REGION Network 3: PID-Pump_1
   #_w1 := "PID_State_Param".PID_Pump1.bModeActivate AND NOT "2_MTrig";   // rising edge
   "2_MTrig" := "PID_State_Param".PID_Pump1.bModeActivate;
   "PID_Compact_Pump-1"(Setpoint := "DB2_HMI_SET"."rSetPump-1_OUT",   // PID_Compact
                        Input := "AI_DB".PT_01.rAI_Value,
                        Reset := NOT "bStartWork_Main",
                        ModeActivate := #_w1,
                        Mode := "PID_State_Param".PID_Pump1.iModeNum,
                        Output => "Pumps".Pump_1.rAutoSpeedPump,
                        State => "PID_State_Param".PID_Pump1.iOutState,
                        Error => "PID_State_Param".PID_Pump1.bOutError,
                        ErrorBits => "PID_State_Param".PID_Pump1.iOutErrorBits);
END_REGION

REGION Network 4 (SCL): Выбор уставки для ПИД насоса - 1
   REGION Parameters PID

      // "PID_Compact_Pump-1".Config.InvertControl := TRUE;

   (* "PID_Compact_Zone1".sRet.r_Ctrl_Gain := "DB2_HMI_SET".k_PID_Zona1.Gain; // Изменение коэф. П
    "PID_Compact_Zone1".sRet.r_Ctrl_Ti  := "DB2_HMI_SET".k_PID_Zona1.I; // Изменение коэф И
    "PID_Compact_Zone1".sRet.r_Ctrl_Td  := "DB2_HMI_SET".k_PID_Zona1.D; // Изменение коэф Д
    *)
    // % Reading Tuning process
       "PID_State_Param".PID_Pump1.iProgress := "PID_Compact_Pump-1".Progress;
   END_REGION



   //Передача уставки в ПИД в зависимости от выбранного режима работы
   IF "bPosition_Diarator" THEN
       "DB2_HMI_SET"."rSetPump-1_OUT" := "DB2_HMI_SET"."rSetPump-1_Diarator";
   ELSE
       "DB2_HMI_SET"."rSetPump-1_OUT" := "DB2_HMI_SET"."rSetPump-1_CIP";
   END_IF;
END_REGION

REGION Network 5: ПИД - насос 2
   #_w1 := "PID_State_Param".PID_Pump2.bModeActivate AND NOT "3_MTrig";   // rising edge
   "3_MTrig" := "PID_State_Param".PID_Pump2.bModeActivate;
   "PID_Compact_Pump-2"(Setpoint := "DB2_HMI_SET"."rSetPump-2_OUT",   // PID_Compact
                        Input := "AI_DB".PT_03.rAI_Value,
                        Reset := NOT "bStartWork_Main",
                        ModeActivate := #_w1,
                        Mode := "PID_State_Param".PID_Pump2.iModeNum,
                        Output => "Pumps".Pump_2.rAutoSpeedPump,
                        State => "PID_State_Param".PID_Pump2.iOutState,
                        Error => "PID_State_Param".PID_Pump2.bOutError,
                        ErrorBits => "PID_State_Param".PID_Pump2.iOutErrorBits);
END_REGION

REGION Network 6 (SCL): Выбор уставки для ПИД насоса - 2
   REGION Parameters PID
       (*"
    PID_Compact_Valve_2".sPid_Cmpt.b_InvCtrl := "bTypePID_Zone1";
    "PID_Compact_Zone1".sRet.r_Ctrl_Gain := "DB2_HMI_SET".k_PID_Zona1.Gain; // Изменение коэф. П
    "PID_Compact_Zone1".sRet.r_Ctrl_Ti  := "DB2_HMI_SET".k_PID_Zona1.I; // Изменение коэф И
    "PID_Compact_Zone1".sRet.r_Ctrl_Td  := "DB2_HMI_SET".k_PID_Zona1.D; // Изменение коэф Д
    *)
    // % Reading Tuning process

   END_REGION
   "PID_State_Param".PID_Pump2.iProgress := "PID_Compact_Pump-2".Progress;
   //Передача уставки в ПИД в зависимости от выбранного режима работы
   IF "bPosition_Diarator" THEN
       "DB2_HMI_SET"."rSetPump-2_OUT" := "DB2_HMI_SET"."rSetPump-2_Diarator";
   ELSE
       "DB2_HMI_SET"."rSetPump-2_OUT" := "DB2_HMI_SET"."rSetPump-2_CIP";
   END_IF;
END_REGION
END_ORGANIZATION_BLOCK

ORGANIZATION_BLOCK "Cyclic interrupt(SCL)"   // OB32, SCL, CyclicInterrupt
{ S7_Optimized_Access := 'TRUE' }
VERSION : 0.1
   VAR_INPUT
      Initial_Call : Bool;   // Initial call of this OB
      Event_Count : Int;   // Events discarded
   END_VAR
   VAR_TEMP
      Reset : Bool;   // Сброс счетчика
   END_VAR
BEGIN
   //Условие включения накопления времени наработки установки (в свойствах ОВ - запуск каждую 1 секунду)
   //Если установка запущена и расход воды больше 1000
   //
   IF "bStartWork_Main" AND "AI_DB".FIC.rAI_Value > 500 THEN
       "diAccumTime" := "diAccumTime" + 1;     // 1 - 1 секунда, запуск ОВ жестко прописан в свойствах ОВ
   END_IF;

   //При необходимости сбросить наккопленную наработку
   //
   "R_trig_ResTimeWorkSystem"(In:="bResTimeWorkSystem",
                              Q=>#Reset);

   IF #Reset THEN
       "diAccumTime" := 0;
   END_IF;

   //Перевод накопленного времени в часы, минуты, секунды
       "iOurs_WorkSystem" := "diAccumTime" / 3600;
       "iMini_WorkSystem" := ("diAccumTime" MOD 3600) / 60;
       "iSec_WorkSystem" := "diAccumTime" MOD 60;
END_ORGANIZATION_BLOCK

ORGANIZATION_BLOCK "Исполнительные устройств"   // OB123, LAD, ProgramCycle
TITLE = Работа физических устройств
{ S7_Optimized_Access := 'TRUE' }
VERSION : 0.1
// Насосы, клапана, и т.д.
   VAR_INPUT
      Initial_Call : Bool;   // Initial call of this OB
      Remanence : Bool;   // =True, if remanent data are available
   END_VAR
BEGIN

REGION Network 1: Аналогвые датчики
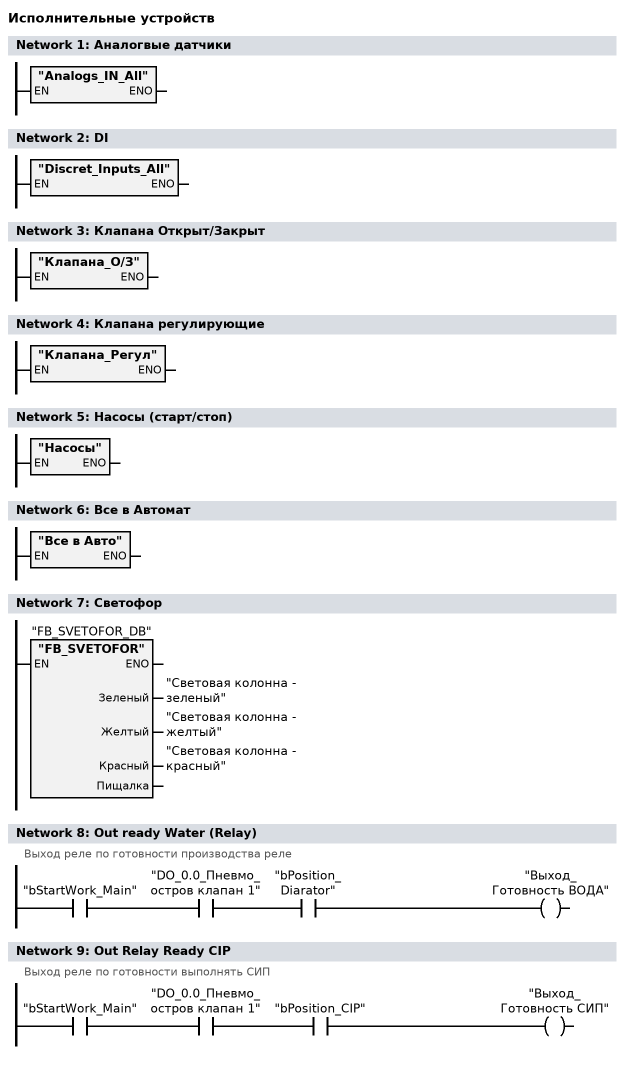
   RUNG wire#powerrail
      "Analogs_IN_All"()
   END_RUNG
   // the same network as SCL:
   "Analogs_IN_All"();
END_REGION

REGION Network 2: DI
   RUNG wire#powerrail
      "Discret_Inputs_All"()
   END_RUNG
   // the same network as SCL:
   "Discret_Inputs_All"();
END_REGION

REGION Network 3: Клапана Открыт/Закрыт
   RUNG wire#powerrail
      "Клапана_О/З"()
   END_RUNG
   // the same network as SCL:
   "Клапана_О/З"();
END_REGION

REGION Network 4: Клапана регулирующие
   RUNG wire#powerrail
      "Клапана_Регул"()
   END_RUNG
   // the same network as SCL:
   "Клапана_Регул"();
END_REGION

REGION Network 5: Насосы (старт/стоп)
   RUNG wire#powerrail
      "Насосы"()
   END_RUNG
   // the same network as SCL:
   "Насосы"();
END_REGION

REGION Network 6: Все в Автомат
   RUNG wire#powerrail
      "Все в Авто"()
   END_RUNG
   // the same network as SCL:
   "Все в Авто"();
END_REGION

REGION Network 7: Светофор
   RUNG wire#powerrail
      "FB_SVETOFOR_DB"(Зеленый => "Световая колонна - зеленый", Желтый => "Световая колонна - желтый", Красный => "Световая колонна - красный", Пищалка =>)
   END_RUNG
   // the same network as SCL:
   "FB_SVETOFOR_DB"(Зеленый => "Световая колонна - зеленый",   // "FB_SVETOFOR"
                    Желтый => "Световая колонна - желтый",
                    Красный => "Световая колонна - красный");
END_REGION

REGION Network 8: Out ready Water (Relay)
   // Выход реле по готовности производства реле
   RUNG wire#powerrail
      Contact( "bStartWork_Main" )
      Contact( "DO_0.0_Пневмо_остров клапан 1" )
      Contact( "bPosition_Diarator" )
      Coil( "Выход_Готовность ВОДА" )
   END_RUNG
   // the same network as SCL:
   "Выход_Готовность ВОДА" := "bStartWork_Main" AND "DO_0.0_Пневмо_остров клапан 1" AND "bPosition_Diarator";
END_REGION

REGION Network 9: Out Relay Ready CIP
   // Выход реле по готовности выполнять СИП
   RUNG wire#powerrail
      Contact( "bStartWork_Main" )
      Contact( "DO_0.0_Пневмо_остров клапан 1" )
      Contact( "bPosition_CIP" )
      Coil( "Выход_Готовность СИП" )
   END_RUNG
   // the same network as SCL:
   "Выход_Готовность СИП" := "bStartWork_Main" AND "DO_0.0_Пневмо_остров клапан 1" AND "bPosition_CIP";
END_REGION
END_ORGANIZATION_BLOCK

ORGANIZATION_BLOCK "Counters"   // OB125, LAD, ProgramCycle
TITLE = "Main Program Sweep (Cycle)"
{ S7_Optimized_Access := 'TRUE' }
VERSION : 0.1
// Различные счетчики
   VAR_INPUT
      Initial_Call : Bool;   // Initial call of this OB
      Remanence : Bool;   // =True, if remanent data are available
   END_VAR
   VAR_TEMP   // added for the SCL form of the ladder/FBD networks
      _w1 : Bool;
      _w2 : Bool;
   END_VAR
BEGIN

REGION Network 1: Counter Water to Sewerage
   // Счетчик сброшенной воды в канализацию
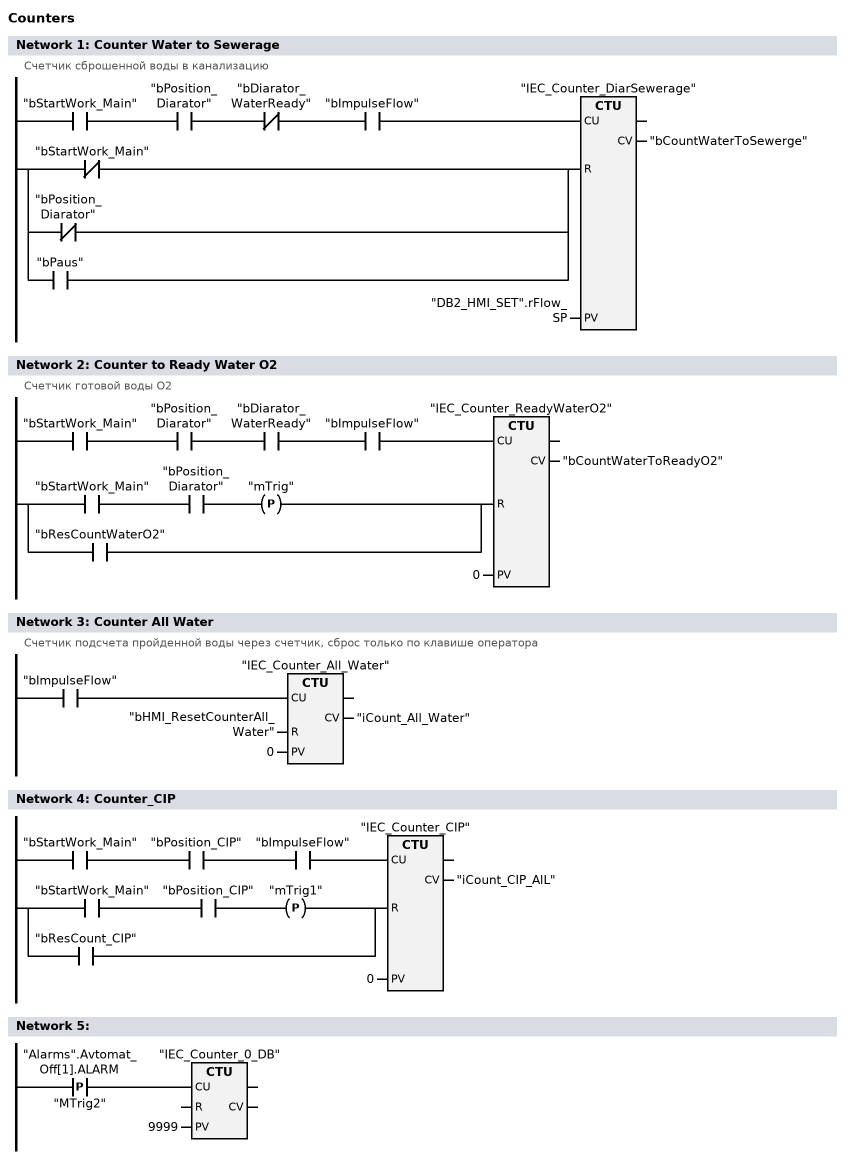
   "IEC_Counter_DiarSewerage".CTU(CU := "bStartWork_Main" AND "bPosition_Diarator" AND NOT "bDiarator_WaterReady" AND "bImpulseFlow",
                           R := NOT "bStartWork_Main" OR NOT "bPosition_Diarator" OR "bPaus",
                           PV := "DB2_HMI_SET".rFlow_SP,
                           CV => "bCountWaterToSewerge");
END_REGION

REGION Network 2: Counter to Ready Water O2
   // Счетчик готовой воды О2
   #_w1 := "bStartWork_Main" AND "bPosition_Diarator";
   #_w2 := #_w1 AND NOT "mTrig";   // rising edge
   "mTrig" := #_w1;
   "IEC_Counter_ReadyWaterO2".CTU(CU := "bStartWork_Main" AND "bPosition_Diarator" AND "bDiarator_WaterReady" AND "bImpulseFlow",
                           R := #_w2 OR "bResCountWaterO2",
                           PV := 0,
                           CV => "bCountWaterToReadyO2");
END_REGION

REGION Network 3: Counter All Water
   // Счетчик подсчета пройденной воды через счетчик, сброс только по клавише оператора
   "IEC_Counter_All_Water".CTU(CU := "bImpulseFlow",
                           R := "bHMI_ResetCounterAll_Water",
                           PV := 0,
                           CV => "iCount_All_Water");
END_REGION

REGION Network 4: Counter_CIP
   #_w1 := "bStartWork_Main" AND "bPosition_CIP";
   #_w2 := #_w1 AND NOT "mTrig1";   // rising edge
   "mTrig1" := #_w1;
   "IEC_Counter_CIP".CTU(CU := "bStartWork_Main" AND "bPosition_CIP" AND "bImpulseFlow",
                         R := #_w2 OR "bResCount_CIP",
                         PV := 0,
                         CV => "iCount_CIP_AlL");
END_REGION

REGION Network 5
   #_w1 := "Alarms".Avtomat_Off[1].ALARM AND NOT "MTrig2";   // rising edge of "Alarms".Avtomat_Off[1].ALARM
   "MTrig2" := "Alarms".Avtomat_Off[1].ALARM;
   "IEC_Counter_0_DB".CTU(CU := #_w1, PV := 9999);
END_REGION
END_ORGANIZATION_BLOCK

// folder: AI_Signal

FUNCTION_BLOCK "AI_(4-20)_1"   // FB13, LAD
{ S7_Optimized_Access := 'FALSE' }
VERSION : 0.1
   VAR_INPUT
      Input_PLC : Int;   // Вход_Значение на ПЛК
      "HMI_Simulate_on/off" : Bool;   // 0 - выкл, 1 - вкл
      HMI_rSimulate_value : Real;   // значение
      HMI_rParam_Sensor_HL : Real := 16.0;   // Параметры датчика по паспорту (макс значение)bar, C, итд
      HMI_rParam_Sensor_LL : Real;   // Параметры датчика по паспорту (мин значение)bar, C, итд
      "HMI_Filtr_On/off" : Bool;   // Фильтрация, true - вкл
   END_VAR
   VAR_OUTPUT
      HMI_Value_OUT : Real;   // Значение в ед. измерения
      Error_out : Bool;   // Ошибка датчика
   END_VAR
   VAR
      OUT_Scale : Real;   // Выход скалированного значения
      OUT_Normal_Ed : Real;   // Выход нормализованной единицы от 0 др 1
      AI_filtr : "AI_Filtr";
      HMI_Range : Int := 10;   // Кол-во данных для фильтрации
      HMI_iSet_Tik : Int := 2;   // Скорость набора данных для фильтрации
   END_VAR
   VAR_TEMP
      Input_PLC_to_dint : DInt;   // Конвертация из инт в реал
      Error : Word;   // Ошибка в скалировании
      "PLC to_real" : Real;
      value_scale : Real;
      Input_PLC_temp : Int;
      OFF_Param : Bool;
   END_VAR
BEGIN

REGION Network 1
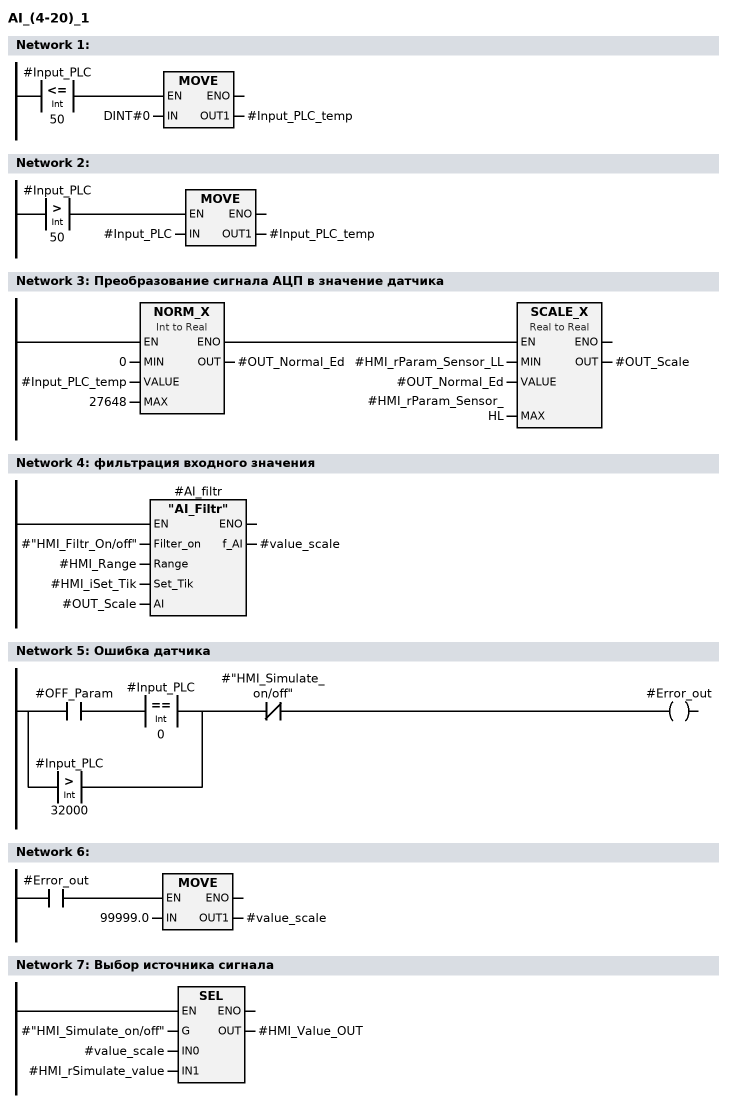
   RUNG wire#powerrail
      { S7_Templates := "SrcType := Int" } LE_Contact(in1 := #Input_PLC, in2 := 50)
      { S7_GenerateENO := "TRUE" } Move(in := DINT#0, out1 => #Input_PLC_temp)
   END_RUNG
   // the same network as SCL:
   IF #Input_PLC <= 50 THEN #Input_PLC_temp := DINT#0; END_IF;
END_REGION

REGION Network 2
   RUNG wire#powerrail
      { S7_Templates := "SrcType := Int" } GT_Contact(in1 := #Input_PLC, in2 := 50)
      { S7_GenerateENO := "TRUE" } Move(in := #Input_PLC, out1 => #Input_PLC_temp)
   END_RUNG
   // the same network as SCL:
   IF #Input_PLC > 50 THEN #Input_PLC_temp := #Input_PLC; END_IF;
END_REGION

REGION Network 3: Преобразование сигнала АЦП в значение датчика
   RUNG wire#powerrail
      { S7_Templates := "[SrcType := Int, DestType := Real]" } Normalize(min := 0, value := #Input_PLC_temp, max := 27648, out => #OUT_Normal_Ed)
      { S7_Templates := "[SrcType := Real, DestType := Real]" } Scale(min := #HMI_rParam_Sensor_LL, value := #OUT_Normal_Ed, max := #HMI_rParam_Sensor_HL, out => #OUT_Scale)
   END_RUNG
   // the same network as SCL:
   #OUT_Normal_Ed := NORM_X(MIN := 0, VALUE := #Input_PLC_temp, MAX := 27648);
   #OUT_Scale := SCALE_X(MIN := #HMI_rParam_Sensor_LL, VALUE := #OUT_Normal_Ed, MAX := #HMI_rParam_Sensor_HL);
END_REGION

REGION Network 4: фильтрация входного значения
   RUNG wire#powerrail
      #AI_filtr(Filter_on := #"HMI_Filtr_On/off", Range := #HMI_Range, Set_Tik := #HMI_iSet_Tik, AI := #OUT_Scale, f_AI => #value_scale)
   END_RUNG
   // the same network as SCL:
   #AI_filtr(Filter_on := #"HMI_Filtr_On/off",   // "AI_Filtr"
             Range := #HMI_Range,
             Set_Tik := #HMI_iSet_Tik,
             AI := #OUT_Scale,
             f_AI => #value_scale);
END_REGION

REGION Network 5: Ошибка датчика
   RUNG wire#powerrail
      Contact( #OFF_Param )
      { S7_Templates := "SrcType := Int" } EQ_Contact(in1 := #Input_PLC, in2 := 0)
      wire#w1
      I_Contact( #"HMI_Simulate_on/off" )
      Coil( #Error_out )
   END_RUNG
   RUNG wire#powerrail
      { S7_Templates := "SrcType := Int" } GT_Contact(in1 := #Input_PLC, in2 := 32000)
   END_RUNG wire#w1
   // the same network as SCL:
   #Error_out := ((#OFF_Param AND (#Input_PLC = 0)) OR (#Input_PLC > 32000)) AND NOT #"HMI_Simulate_on/off";
END_REGION

REGION Network 6
   RUNG wire#powerrail
      Contact( #Error_out )
      Move(in := 99999.0, out1 => #value_scale)
   END_RUNG
   // the same network as SCL:
   IF #Error_out THEN #value_scale := 99999.0; END_IF;
END_REGION

REGION Network 7: Выбор источника сигнала
   #HMI_Value_OUT := SEL(G := #"HMI_Simulate_on/off", IN0 := #value_scale, IN1 := #HMI_rSimulate_value);
END_REGION
END_FUNCTION_BLOCK

FUNCTION_BLOCK "AI_(PT100)"   // FB21, LAD
{ S7_Optimized_Access := 'FALSE' }
VERSION : 0.1
   VAR_INPUT
      Input_PLC : Int;   // Вход_Значение на ПЛК
      "Simulate_on/off" : Bool;   // 0 - выкл, 1 - вкл
      Simulate_value : Real;   // значение
      Param_Sensor_HL : Real := 16.0;   // Параметры датчика по паспорту (макс значение)bar, C, итд
      Param_Sensor_LL : Real;   // Параметры датчика по паспорту (мин значение)bar, C, итд
      "Filtr_On/off" : Bool;   // Фильтрация, true - вкл
   END_VAR
   VAR_OUTPUT
      Value_OUT : Real;   // Значение в ед. измерения
      Error_out : Bool;   // Ошибка датчика
   END_VAR
   VAR
      bipolar : Bool;
      OUT_Scale : Real;   // Выход скалированного значения
      AI_filtr : "AI_Filtr";
      Range : Int := 10;   // Кол-во данных для фильтрации
   END_VAR
   VAR_TEMP
      Input_PLC_to_dint : DInt;   // Конвертация из инт в реал
      Error : Word;   // Ошибка в скалировании
      "PLC to_real" : Real;
      value_scale : Real;
      Input_PLC_temp : Int;
      Input_PLC_to_real : Real;
   END_VAR
BEGIN

REGION Network 1
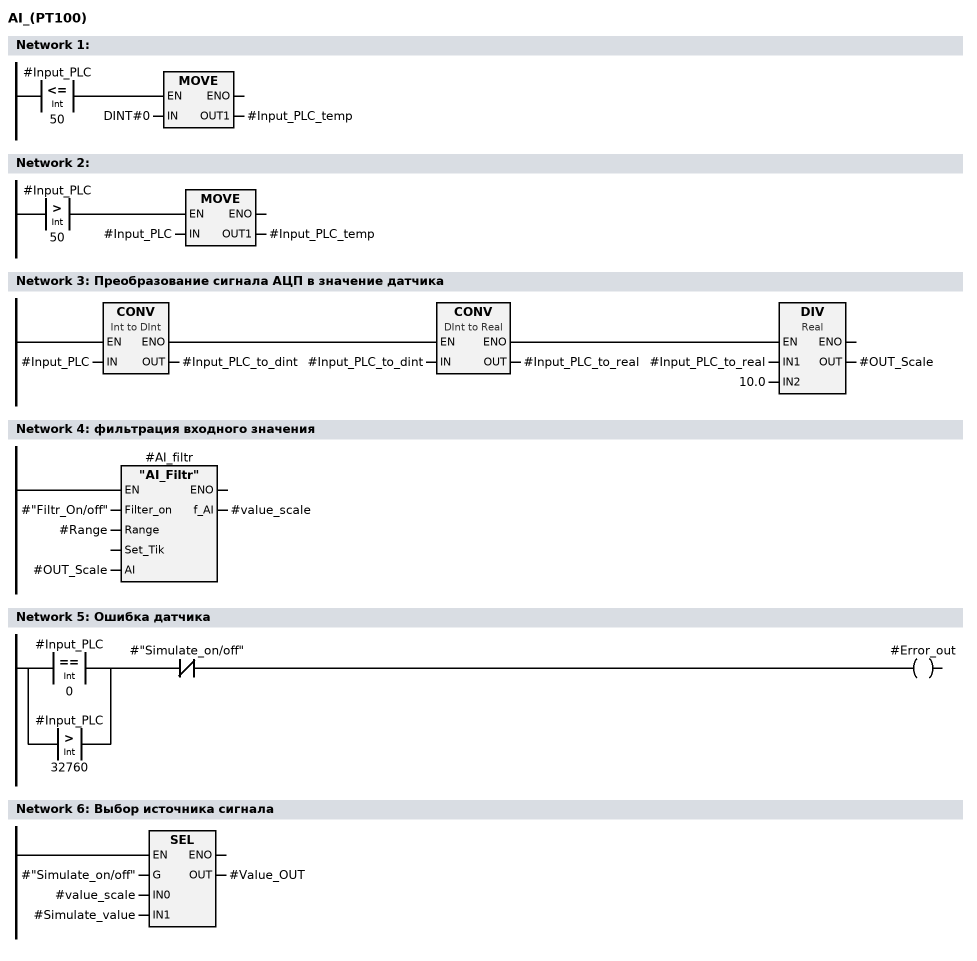
   RUNG wire#powerrail
      { S7_Templates := "SrcType := Int" } LE_Contact(in1 := #Input_PLC, in2 := 50)
      { S7_GenerateENO := "TRUE" } Move(in := DINT#0, out1 => #Input_PLC_temp)
   END_RUNG
   // the same network as SCL:
   IF #Input_PLC <= 50 THEN #Input_PLC_temp := DINT#0; END_IF;
END_REGION

REGION Network 2
   RUNG wire#powerrail
      { S7_Templates := "SrcType := Int" } GT_Contact(in1 := #Input_PLC, in2 := 50)
      { S7_GenerateENO := "TRUE" } Move(in := #Input_PLC, out1 => #Input_PLC_temp)
   END_RUNG
   // the same network as SCL:
   IF #Input_PLC > 50 THEN #Input_PLC_temp := #Input_PLC; END_IF;
END_REGION

REGION Network 3: Преобразование сигнала АЦП в значение датчика
   RUNG wire#powerrail
      { S7_Templates := "[SrcType := Int, DestType := DInt]"; S7_GenerateENO := "TRUE" } Convert(in := #Input_PLC, out => #Input_PLC_to_dint)
      { S7_Templates := "[SrcType := DInt, DestType := Real]"; S7_GenerateENO := "TRUE" } Convert(in := #Input_PLC_to_dint, out => #Input_PLC_to_real)
      { S7_Templates := "SrcType := Real"; S7_GenerateENO := "TRUE" } Div(in1 := #Input_PLC_to_real, in2 := 10.0, out => #OUT_Scale)
   END_RUNG
   // the same network as SCL:
   // ENO of a box is taken as its EN; it also drops when the box reports an error
   #Input_PLC_to_dint := INT_TO_DINT(#Input_PLC);
   #Input_PLC_to_real := DINT_TO_REAL(#Input_PLC_to_dint);
   #OUT_Scale := #Input_PLC_to_real / 10.0;
END_REGION

REGION Network 4: фильтрация входного значения
   RUNG wire#powerrail
      #AI_filtr(Filter_on := #"Filtr_On/off", Range := #Range, Set_Tik :=, AI := #OUT_Scale, f_AI => #value_scale)
   END_RUNG
   // the same network as SCL:
   #AI_filtr(Filter_on := #"Filtr_On/off", Range := #Range, AI := #OUT_Scale, f_AI => #value_scale);   // "AI_Filtr"
END_REGION

REGION Network 5: Ошибка датчика
   RUNG wire#powerrail
      { S7_Templates := "SrcType := Int" } EQ_Contact(in1 := #Input_PLC, in2 := 0)
      wire#w1
      I_Contact( #"Simulate_on/off" )
      Coil( #Error_out )
   END_RUNG
   RUNG wire#powerrail
      { S7_Templates := "SrcType := Int" } GT_Contact(in1 := #Input_PLC, in2 := 32760)
   END_RUNG wire#w1
   // the same network as SCL:
   #Error_out := ((#Input_PLC = 0) OR (#Input_PLC > 32760)) AND NOT #"Simulate_on/off";
END_REGION

REGION Network 6: Выбор источника сигнала
   #Value_OUT := SEL(G := #"Simulate_on/off", IN0 := #value_scale, IN1 := #Simulate_value);
END_REGION
END_FUNCTION_BLOCK

// folder: AI_Signal/Funktion

FUNCTION_BLOCK "AI_Filtr"   // FB14, SCL
{ S7_Optimized_Access := 'FALSE' }
VERSION : 0.1
   VAR_INPUT
      Filter_on : Bool;   // Вкл фильтрации
      Range : Int := 10;   // Кол-во входных значений для вычисления среднего
      Set_Tik : Int := 6;   // Задача периода фильтрации от 1(мин) до 8
      AI : Real;   // Вход значения датчика
   END_VAR
   VAR_OUTPUT
      f_AI : Real;   // выход значения с фильтром или без
   END_VAR
   VAR
      CTU : CTU_INT;   // счетчик для подсчета кол-во вх значений
      Tik : Bool;   // Время фильтрации
      ai_array : Array[0..#Max_Array] of Real;   // Массив значений датчика
      i : Int;   // для цикла ФОР
      sum_AI : Real;   // Суммирование значений с входа датчика
      Avarage_AI : Real;   // Среднее значение датчика
      fRS_set : Bool;   // Для RS тригера
      fRS_res : Bool;   // Для RS тригера
      fRS_out : Bool;   // Для RS тригера
      FullFiltr : Bool;   // Ожидание наполнения значений для вычисления средней
      Res_count : Bool;   // сброс счетчика
   END_VAR
   VAR CONSTANT
      Max_Array : Int := 30;   // Размер массива
   END_VAR
BEGIN

   CASE #Set_Tik OF                   
       1:  
           #Tik := "Time_0.1s";
       2:  
           #Tik := "Time_0.2s";
       3:
           #Tik := "Time_0.4s";
       4:
           #Tik := "Time_0.5s";
       5:
           #Tik := "Time_0.8s";
       6:
           #Tik := "Time_1s";
       7:
           #Tik := "Time_1.6s";
       8:
           #Tik := "Time_2s";
       0:
           #Tik := "Time_0.1s";

       ELSE  
           #Set_Tik := 8;
   END_CASE;  // Выбор периода фильтрации входного сигнала
   REGION RS триггер
       IF #fRS_set THEN
           #fRS_out := true;
       ELSIF #fRS_res AND NOT #fRS_set THEN
           #fRS_out := false;
       END_IF;
   END_REGION

   REGION Подсчет среднего значения входа
       // Statement section REGION
           #CTU(CU := #Tik,
                PV := #Range,
                R := #Res_count,
                Q => #Res_count);                                      // Счетчик для набора значений с входа
           #ai_array[#CTU.CV] := #AI;                                  // Запись значений с входа в массив

           IF #Res_count THEN                                              // СБРОС как счетчик переполниться Для корректной работы счетчика
               #i := 0;
               #sum_AI := 0;
           END_IF;

           IF #Range <> #i THEN                                    // выход из цикла FOR при суммировании всех значений, почему то сам не прекращел подсчет при окончании цикла все время суммировался 
               FOR #i := 0 TO (#Range - 1) DO
                   #sum_AI := #ai_array[#i] + #sum_AI;             // суммирование значений
               END_FOR;
           END_IF;

       #Avarage_AI := #sum_AI / #Range;                             // Вычисление среднего значения
       #fRS_res := NOT #Filter_on;

   END_REGION

   REGION Выбор выхода прямое или фильтрованное значение
       IF #Filter_on THEN                                          //Включение выключение фильтрации
           #fRS_set := #CTU.QD;                                    //При включении фильтра ждем наполнения значениями с входа, пока ждем - отправляем на выход прямое значение входа, далее фильтруем
            #FullFiltr := #fRS_out;

          IF #FullFiltr THEN                                       //Когда фильтр наполнился - вывыодим среднее значение входа
               #f_AI := #Avarage_AI;                              // ЗАпись значения на выход AI
          ELSE
               #f_AI := #AI;                                     // Прямой вывод значения, пока значения не наполнились данными
          END_IF;
       ELSE
           #f_AI := #AI;                                        // Если фильтр выключен, на выход прямое значение с входа
       END_IF; 

   END_REGION
END_FUNCTION_BLOCK

FUNCTION "Calculate_AI" : Void   // FC7, SCL
{ S7_Optimized_Access := 'FALSE' }
VERSION : 0.1
   VAR_INPUT
      IN_sensors : Int;
      Current_max : Real;
      Current_min : Real;
      Code_HL : Real;
      Code_LL : Real;
      Param_Sensor_HL : Real;   // Параметры датчика по паспорту (макс значение)bar, C, итд
      Param_Sensor_LL : Real;   // Параметры датчика по паспорту (мин значение)bar, C, итд
   END_VAR
   VAR_OUTPUT
      signal_Electric : Real;   // выход в электрических ед измерения
      Value_Sensor : Real;   // выход реального значения датчика в ед измерения
   END_VAR
   VAR_TEMP
      sensor_to_real : Real;   // Для конвертации INT to Real
      result_to_out_signal : Real;   // Для вычитания реального значения показания датчика
   END_VAR
BEGIN
       //Convert int to real
   #sensor_to_real := INT_TO_REAL(#IN_sensors);

       // Расчет значения АЦП контроллера в значение эл. ед измерения (I, U) в зависимости от значений на входе
   #signal_Electric := ((#sensor_to_real - #Code_LL) * (#Current_max - #Current_min) / (#Code_HL - #Code_LL))+ #Current_min;
   #result_to_out_signal := #signal_Electric;

   // Расчет значения в реальных единицах измерения датчика (bar, C,) в зависимости от введеных параметров датчика Param_Sensor min/max
   #Value_Sensor := (#result_to_out_signal - #Current_min) * (#Param_Sensor_HL - #Param_Sensor_LL) / (#Current_max - #Current_min) + #Param_Sensor_LL;
END_FUNCTION

// folder: DI_signal

FUNCTION_BLOCK "FB_DI"   // FB15, LAD
TITLE = Блок обработки дискретных входов
{ S7_Optimized_Access := 'FALSE' }
VERSION : 0.1
   VAR_INPUT
      input_value : Bool;   // Входной тэг контроллера
      "On/Off_Filters_DI" : Bool;   // Вкл/выкл фильтрацию входа
      Set_Time_Dely : Time;   // Уставка времени фильтрации
      Simulate : Bool;   // Симуляция входа (Вкл/Выкл)
      Simulate_Value : Bool;   // Значение симуляции
   END_VAR
   VAR_OUTPUT
      Value : Bool;   // Обработанный сигнал
   END_VAR
   VAR
      Time_Delay : Time;   // Время фильтрации для таймера
      Time_On : TON_TIME;   // Фильтр на Вкл
      Time_Off : TON_TIME;   // Фильтр на Выкл
      Nul_Time : Time := T#1MS;   // Откл фильтрации (0)
   END_VAR
BEGIN

REGION Network 1: Включение фильтрации
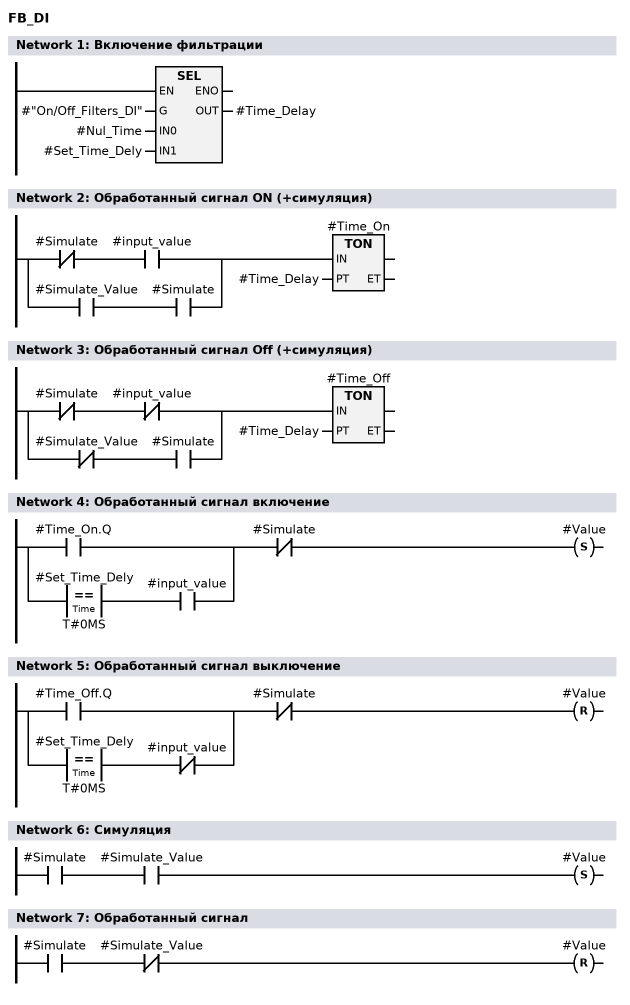
   #Time_Delay := SEL(G := #"On/Off_Filters_DI", IN0 := #Nul_Time, IN1 := #Set_Time_Dely);
END_REGION

REGION Network 2: Обработанный сигнал ON (+симуляция)
   #Time_On(IN := (NOT #Simulate AND #input_value) OR (#Simulate_Value AND #Simulate), PT := #Time_Delay);   // TON
END_REGION

REGION Network 3: Обработанный сигнал Off (+симуляция)
   #Time_Off(IN := (NOT #Simulate AND NOT #input_value) OR (NOT #Simulate_Value AND #Simulate),   // TON
             PT := #Time_Delay);
END_REGION

REGION Network 4: Обработанный сигнал включение
   RUNG wire#powerrail
      Contact( #Time_On.Q )
      wire#w1
      I_Contact( #Simulate )
      S_Coil( #Value )
   END_RUNG
   RUNG wire#powerrail
      { S7_Templates := "SrcType := Time" } EQ_Contact(in1 := #Set_Time_Dely, in2 := T#0MS)
      Contact( #input_value )
   END_RUNG wire#w1
   // the same network as SCL:
   IF (#Time_On.Q OR ((#Set_Time_Dely = T#0MS) AND #input_value)) AND NOT #Simulate THEN
       #Value := TRUE;
   END_IF;
END_REGION

REGION Network 5: Обработанный сигнал выключение
   RUNG wire#powerrail
      Contact( #Time_Off.Q )
      wire#w1
      I_Contact( #Simulate )
      R_Coil( #Value )
   END_RUNG
   RUNG wire#powerrail
      { S7_Templates := "SrcType := Time" } EQ_Contact(in1 := #Set_Time_Dely, in2 := T#0MS)
      I_Contact( #input_value )
   END_RUNG wire#w1
   // the same network as SCL:
   IF (#Time_Off.Q OR ((#Set_Time_Dely = T#0MS) AND NOT #input_value)) AND NOT #Simulate THEN
       #Value := FALSE;
   END_IF;
END_REGION

REGION Network 6: Симуляция
   RUNG wire#powerrail
      Contact( #Simulate )
      Contact( #Simulate_Value )
      S_Coil( #Value )
   END_RUNG
   // the same network as SCL:
   IF #Simulate AND #Simulate_Value THEN #Value := TRUE; END_IF;
END_REGION

REGION Network 7: Обработанный сигнал
   RUNG wire#powerrail
      Contact( #Simulate )
      I_Contact( #Simulate_Value )
      R_Coil( #Value )
   END_RUNG
   // the same network as SCL:
   IF #Simulate AND NOT #Simulate_Value THEN #Value := FALSE; END_IF;
END_REGION
END_FUNCTION_BLOCK

FUNCTION_BLOCK "FB_DI_Pointer"   // FB17, LAD
TITLE = Блок обработки дискретных входов
{ S7_Optimized_Access := 'FALSE' }
VERSION : 0.1
   VAR_INPUT
      input_value : Bool;   // Входной тэг контроллера
   END_VAR
   VAR_OUTPUT
      Value : Bool;   // Обработанный сигнал
   END_VAR
   VAR_IN_OUT
      Di_Struct : "Tipe_DI";
   END_VAR
   VAR
      Time_Delay : Time;   // Время фильтрации для таймера
      Time_On : TON_TIME;   // Фильтр на Вкл
      Time_Off : TON_TIME;   // Фильтр на Выкл
      Nul_Time : Time := T#1MS;   // Откл фильтрации (0)
      testdel : Bool;
      On_del : Bool;
   END_VAR
BEGIN

REGION Network 1: Включение фильтрации
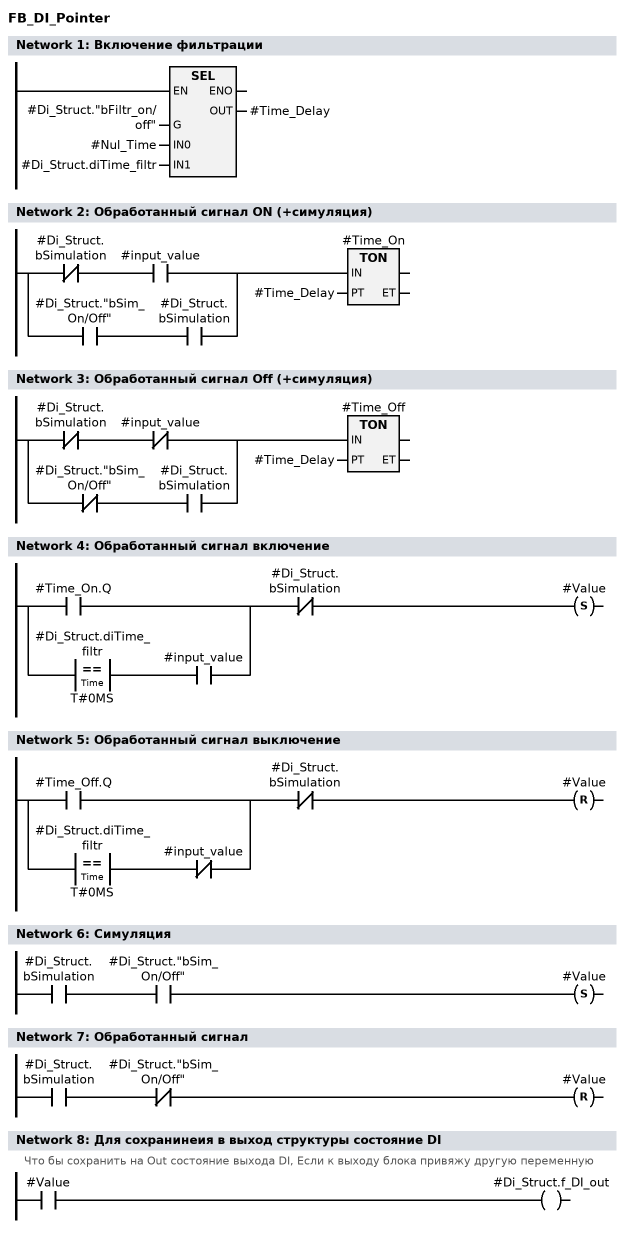
   #Time_Delay := SEL(G := #Di_Struct."bFiltr_on/off", IN0 := #Nul_Time, IN1 := #Di_Struct.diTime_filtr);
END_REGION

REGION Network 2: Обработанный сигнал ON (+симуляция)
   #Time_On(IN := (NOT #Di_Struct.bSimulation AND #input_value) OR (#Di_Struct."bSim_On/Off" AND #Di_Struct.bSimulation),   // TON
            PT := #Time_Delay);
END_REGION

REGION Network 3: Обработанный сигнал Off (+симуляция)
   #Time_Off(IN := (NOT #Di_Struct.bSimulation AND NOT #input_value) OR (NOT #Di_Struct."bSim_On/Off" AND #Di_Struct.bSimulation),   // TON
             PT := #Time_Delay);
END_REGION

REGION Network 4: Обработанный сигнал включение
   RUNG wire#powerrail
      Contact( #Time_On.Q )
      wire#w1
      I_Contact( #Di_Struct.bSimulation )
      S_Coil( #Value )
   END_RUNG
   RUNG wire#powerrail
      { S7_Templates := "SrcType := Time" } EQ_Contact(in1 := #Di_Struct.diTime_filtr, in2 := T#0MS)
      Contact( #input_value )
   END_RUNG wire#w1
   // the same network as SCL:
   IF (#Time_On.Q OR ((#Di_Struct.diTime_filtr = T#0MS) AND #input_value)) AND NOT #Di_Struct.bSimulation THEN
       #Value := TRUE;
   END_IF;
END_REGION

REGION Network 5: Обработанный сигнал выключение
   RUNG wire#powerrail
      Contact( #Time_Off.Q )
      wire#w1
      I_Contact( #Di_Struct.bSimulation )
      R_Coil( #Value )
   END_RUNG
   RUNG wire#powerrail
      { S7_Templates := "SrcType := Time" } EQ_Contact(in1 := #Di_Struct.diTime_filtr, in2 := T#0MS)
      I_Contact( #input_value )
   END_RUNG wire#w1
   // the same network as SCL:
   IF (#Time_Off.Q OR ((#Di_Struct.diTime_filtr = T#0MS) AND NOT #input_value)) AND NOT #Di_Struct.bSimulation THEN
       #Value := FALSE;
   END_IF;
END_REGION

REGION Network 6: Симуляция
   RUNG wire#powerrail
      Contact( #Di_Struct.bSimulation )
      Contact( #Di_Struct."bSim_On/Off" )
      S_Coil( #Value )
   END_RUNG
   // the same network as SCL:
   IF #Di_Struct.bSimulation AND #Di_Struct."bSim_On/Off" THEN #Value := TRUE; END_IF;
END_REGION

REGION Network 7: Обработанный сигнал
   RUNG wire#powerrail
      Contact( #Di_Struct.bSimulation )
      I_Contact( #Di_Struct."bSim_On/Off" )
      R_Coil( #Value )
   END_RUNG
   // the same network as SCL:
   IF #Di_Struct.bSimulation AND NOT #Di_Struct."bSim_On/Off" THEN #Value := FALSE; END_IF;
END_REGION

REGION Network 8: Для сохранинеия в выход структуры состояние DI
   // Что бы сохранить на Out состояние выхода DI, Если к выходу блока привяжу другую переменную
   RUNG wire#powerrail
      Contact( #Value )
      Coil( #Di_Struct.f_DI_out )
   END_RUNG
   // the same network as SCL:
   #Di_Struct.f_DI_out := #Value;
END_REGION
END_FUNCTION_BLOCK

// folder: FB

FUNCTION_BLOCK "R_trig"   // FB16, SCL
{ S7_Optimized_Access := 'TRUE' }
VERSION : 0.1
   VAR_INPUT
      In : Bool;
   END_VAR
   VAR_OUTPUT
      Q : Bool;
   END_VAR
   VAR
      Click_M : Bool;
   END_VAR
BEGIN
   #Q := #In AND NOT #Click_M;
   #Click_M := #In;
END_FUNCTION_BLOCK

// folder: FB_Elemets

FUNCTION_BLOCK "Pump"   // FB1, SCL
{ S7_Optimized_Access := 'FALSE' }
VERSION : 0.1
   VAR_INPUT
      bManualMode : Bool;   // Выбор ручного режима
      bManualStart : Bool;   // Ручной режим - старт
      bManualStop : Bool;   // Ручной режим - стоп
      rManualSpeed : Real;   // Ручной режим - скорость
      bDryRunn : Bool;   // Защита от сухого хода, False - сухой ход
      bAutoSTop : Bool;   // Остановка насоса
      bAutoStartPerm : Bool;   // Команда на работоу в авто режиме
      rAutoSpeed : Real;   // Скорость в авто режиме
      bАвтоматы : Bool;   // Готовность привода (автоматы)
      bПускатели : Bool;   // Готовность Пускателя
      bDriveRunning : Bool;   // Привод в работе
      bDriveFault : Bool;   // Привод в ошибке
      rMinSpeed : Real;   // Минимальная скорость
      rMaxSpeed : Real := 100.0;   // Максимальная скорость
      bResetFault : Bool;   // Сброс аварии
   END_VAR
   VAR_OUTPUT
      bRunCmd : Bool;   // Пуск частотника
      iSpeedOut : Int;   // Скорость насоса для аналогового выхода
      "rSpeedHMI(0-100)" : Real;   // Скорость работы (0-100) для HMI
      bPumpRunning : Bool;   // Работа
      bPumpFault : Bool;   // Авария
      iStatus : Int;   // Статус (0 - стоп 1 - работа 2 - авария)
   END_VAR
   VAR
      bFaultLatch : Bool;
      bRunRequest : Bool;
      rSpeedPump : Real;   // Скорость насоса
      TON_NotStartRun : TON_TIME;   // ТАймер ожидания сигнала о запуске
      TON_NotContactRun : TON_TIME;   // ТАймер ожидания с контактора
      TON_DryStop : TON_TIME;   // Стоп оп сухому ходу
      TON_DryRun : TON_TIME;   // Таймер старт после появления сигнала сухого хода
   END_VAR
BEGIN
   (*
   // 1. Обработка аварий
   // Обработка ожидания сигнала о работе после старта
   IF #bAutoStartPerm THEN
       ;

   END_IF;
   *)

   // 1 Ручной режим
   IF #bManualMode THEN
       // Ручной режим
       IF #bManualStart AND NOT #bManualStop THEN
           #bRunRequest := TRUE;
       ELSIF #bManualStop THEN // OR NOT #bАвтоматы THEN
           #bRunRequest := FALSE;
       END_IF;
   ELSE
       // Автоматический режим
       // 
       //Обработка аварий
       //--------------------------------------------------------------------------------------------------------
       IF #bAutoStartPerm AND NOT #bAutoSTop THEN
           #TON_NotStartRun(IN := NOT #bDriveRunning AND #bDryRunn,
                            PT := t#5s);  //Таймер ожидания сигнала подтверждения пуска от частотника
           #TON_NotContactRun(IN := NOT #bПускатели,
                              PT := t#5s);  //Таймер ожидания сигнала подтверждения пуска от пускателя
           #TON_DryRun(IN := #bDryRunn,
                       PT := t#2s);    //Таймер ожидания старта после поялвения сигнала по сухому ходу
           #TON_DryStop(IN := NOT #bDryRunn,
                       PT := t#2s);    //Таймер ожидания старта после поялвения сигнала по сухому ходу

       ELSE
           #TON_NotStartRun(IN := FALSE,
                            PT := t#5s);
           #TON_NotContactRun(IN := FALSE,
                              PT := t#5s);
       END_IF;
       #bFaultLatch := #TON_NotStartRun.Q OR #TON_NotContactRun.Q OR (#bDriveFault OR NOT #bАвтоматы) OR (NOT #bResetFault AND #bFaultLatch); //Разкоментировать если нужна будет фиксация АЛАРМА, сброс только по входу РЕСЕТ
       #bPumpFault := #bFaultLatch;

       //Старт--------------------------------
       IF #bAutoStartPerm AND NOT #bPumpFault AND #TON_DryRun.Q THEN
           #bRunRequest := TRUE;
       ELSIF #bAutoStartPerm AND NOT #bPumpFault AND #TON_DryStop.Q THEN
           #bRunRequest := FALSE;
       END_IF;


   END_IF;

   // 3. Задание скорости
   IF #bManualMode THEN
       #"rSpeedHMI(0-100)" := LIMIT(MN := #rMinSpeed, IN := #rManualSpeed, MX := #rMaxSpeed);
   ELSIF
       NOT #bManualMode AND NOT #bRunCmd THEN
       #"rSpeedHMI(0-100)" := 0;
   ELSE
       #"rSpeedHMI(0-100)" := LIMIT(MN := #rMinSpeed, IN := #rAutoSpeed, MX := #rMaxSpeed);
   END_IF;

   // Преобразование значения от 0-100 до 0-27648 для аналогового выхода
   #iSpeedOut := REAL_TO_INT((#"rSpeedHMI(0-100)" / 100.0) * 27648.0);

   // 4. Выходные команды и статусы
   // Команды старт
   #bRunCmd := #bRunRequest;

   //Выход статуса для HMI
   #bPumpRunning := #bDriveRunning AND #bRunCmd AND NOT #bAutoSTop OR (#bManualMode AND #bRunRequest);



   // 5. Числовой статус (для HMI/SCADA)
   IF #bFaultLatch THEN
       #iStatus := 2; // Авария
   ELSIF #bPumpRunning OR (#bManualMode AND #bRunRequest) THEN
       #iStatus := 1; // Работа
   ELSE
       #iStatus := 0; // Стоп
   END_IF;

   IF #bAutoSTop AND NOT #bManualMode THEN
       #bRunCmd := FALSE;
   END_IF;
   IF #bResetFault THEN
       #bFaultLatch := FALSE;
   END_IF;
END_FUNCTION_BLOCK

FUNCTION_BLOCK "Valve(c/o)"   // FB3, SCL
{ S7_Optimized_Access := 'FALSE' }
VERSION : 0.1
   VAR_INPUT
      bAuto_OpenCmd : Bool;   // Команда открыть (автомат)
      bManualMode : Bool;   // Ручной режим (TRUE)
      bManualOpen : Bool;   // Команда открыть в ручном режиме
      bFeedback : Bool;   // Обратная связь "закрытт"
      tMaxTime : Time;   // Время на открытие
      bResetAlarm : Bool;   // Сброс аварии
      bHaveFeedback : Bool;   // Есть ли обратная связь (0 - нет, 1 есть)
   END_VAR
   VAR_OUTPUT
      bValveOpen : Bool;   // Управляющий выход
      iValveState : Int;   // 0 = Закрыт, 1 = Открыт, 2 = Авария
      bValveFault : Bool;   // Авария
   END_VAR
   VAR
      tiOpenTimer : TON_TIME;   // Таймер на открытие
      bWaitingOpen : Bool;   // Флаг ожидания открытия
      bEnableTimer : Bool;   // Флаг активации таймера
   END_VAR
BEGIN

   // Обновление таймера — всегда в одном месте, вне условий
   #tiOpenTimer(
                IN := #bEnableTimer,
                PT := #tMaxTime *1000
   );

   // Сброс
   IF #bResetAlarm THEN
       #bValveFault := FALSE;
       #bWaitingOpen := FALSE;
       #bEnableTimer := FALSE;
   END_IF;

   // === Режим: РУЧНОЙ ===
   IF #bManualMode THEN
       #bValveOpen := #bManualOpen;
       #bValveFault := FALSE;          // Аварии в ручном режиме не учитываются
       #bEnableTimer := FALSE;
       #bWaitingOpen := FALSE;

       // === Режим: АВТО ===
   ELSE

           // Управление выходом с учетом аварии, с контролем обратной связи
        IF #bAuto_OpenCmd AND NOT #bValveFault THEN
                   #bValveOpen := TRUE;
        ELSE
                   #bValveOpen := FALSE;
               END_IF;

               //  Проверяем, есть ли контроль обратной связи
        IF #bHaveFeedback THEN
            // Контроль открытия
            IF #bAuto_OpenCmd AND #bFeedback AND NOT #bValveFault THEN
                #bEnableTimer := TRUE;
                #bWaitingOpen := TRUE;
            ELSE
                #bEnableTimer := FALSE;
                ;
                IF #bFeedback THEN
                    #bWaitingOpen := FALSE;
                END_IF;
            END_IF;
        END_IF;


           // Авария
           IF #tiOpenTimer.Q AND #bWaitingOpen THEN
               #bValveFault := TRUE;
               #bWaitingOpen := FALSE;
           END_IF;

           IF NOT #bAuto_OpenCmd AND NOT #bFeedback AND #bHaveFeedback THEN
               #bEnableTimer := TRUE;
               #bWaitingOpen := TRUE;
           ELSIF
               #bAuto_OpenCmd AND #bFeedback AND #bHaveFeedback THEN
                   #bEnableTimer := TRUE;
                   #bWaitingOpen := TRUE;        ELSE
               #bEnableTimer := FALSE;
               IF #bFeedback THEN
                   #bWaitingOpen := FALSE;
               END_IF;
           END_IF;

   END_IF;


   // Состояние клапана
   IF #bValveFault THEN
       #iValveState := 2;       // Авария
   ELSIF #bHaveFeedback AND NOT #bFeedback  THEN
       #iValveState := 1;       // Открыт
   ELSIF NOT #bHaveFeedback AND (NOT #bManualMode AND #bAuto_OpenCmd) OR (#bManualOpen AND #bManualMode) THEN
       #iValveState := 1;       // Открыт 
   ELSE
       #iValveState := 0;       // Закрыт
   END_IF;
END_FUNCTION_BLOCK

FUNCTION_BLOCK "Valve(regul)"   // FB4, SCL
{ S7_Optimized_Access := 'FALSE' }
VERSION : 0.1
   VAR_INPUT
      bManualMode : Bool;   // TRUE = ручной режим, FALSE = автоматический режим
      rAutoSetpoint : Real;   // Уставка открытия клапана в % (0.0–100.0) в автомате
      rManualSetpoint : Real;   // Уставка открытия клапана в % (0.0–100.0) в ручном режиме
   END_VAR
   VAR_OUTPUT
      iAnalogOutput : Int;   // Значение для аналогового выхода (0–27648)
      rValvePosPercent : Real;   // Текущее % открытия клапана для HMI
      bValveOpen : Bool;   // Дискретный сигнал "клапан открыт" (TRUE, если >0%)
   END_VAR
   VAR
      rSetpointPercent : Real;   // Расчётная уставка % открытия в текущем режиме
   END_VAR
BEGIN
       // Выбор уставки в зависимости от режима
       IF #bManualMode THEN
           #rSetpointPercent := #rManualSetpoint;
       ELSE
           #rSetpointPercent := #rAutoSetpoint;
       END_IF;

       // Ограничение % от 0.0 до 100.0
       IF #rSetpointPercent < 0.0 THEN
           #rSetpointPercent := 0.0;
       ELSIF #rSetpointPercent > 100.0 THEN
           #rSetpointPercent := 100.0;
       END_IF;

       // Перевод % в значение для аналогового выхода
       #iAnalogOutput := REAL_TO_INT((#rSetpointPercent / 100.0) * 27648.0);

           // Вывод значения для HMI
       #rValvePosPercent := #rSetpointPercent;

       // Дискретный сигнал "клапан открыт", если % > 0
       #bValveOpen := #rSetpointPercent > 0.0;
END_FUNCTION_BLOCK